// Base class for all error classes.
{attribute 'enable_dynamic_creation'}
{attribute 'reflection'}
{attribute 'no_explicit_call' := 'direct call for this function block is not allowed'}
FUNCTION_BLOCK FsFB_Error EXTENDS FsFB_ValueType IMPLEMENTS FsI_Error
VAR
	_Code : FsT_ErrCode := FsGVL_ErrorCodes.NO_ERROR;
	_Message : FsT_ErrMsg := 'No Error.';
END_VAR

PROPERTY Code : FsT_ErrCode
GET
Code := THIS^._Code;
END_GET
END_PROPERTY

PROPERTY PROTECTED DynamicTypeName : FsT_Str
GET
VAR
	fbVar : FsFB_Error;
	VarInfo : FsT_VarInfo := __VARINFO(fbVar); 
END_VAR
DynamicTypeName := VarInfo.TypeName;
END_GET
END_PROPERTY

PROPERTY Message : FsT_ErrSrc
GET
Message := THIS^._Message;
END_GET
END_PROPERTY

END_FUNCTION_BLOCK

(* stored: Version 1.1.0.1, ProductVersion 3.1.4024.4
   POU FsFB_Error: Id {c4eb7949-7443-499c-949e-98da50b3b761}, SpecialFunc None
   Folder Properties: Id {a7b71548-d192-42d0-8705-19b65dcc0eef}
   Property Code: Id {ce1ad6ad-2d4a-457e-b32d-a7a05170f8d1}
   Get Get: Id {ae7a7f3d-3705-4e3b-99fa-7a34c4629ddc}
   Property DynamicTypeName: Id {539e9e46-bc25-4de6-be76-e3d8dfd2e7bb}
   Get Get: Id {5208f2fe-8673-4479-bd9b-5fbfa36beb71}
   Property Message: Id {0275838e-9083-4da7-a021-40525c78aa89}
   Get Get: Id {8abb904a-cc63-4170-a83d-153219f77c65} *)
